# B&R Automation Studio project DuctLines (part 15)

### Program Logical/Uncoiler_2 (IEC)

#### Cyclic.ld - Cyclic code
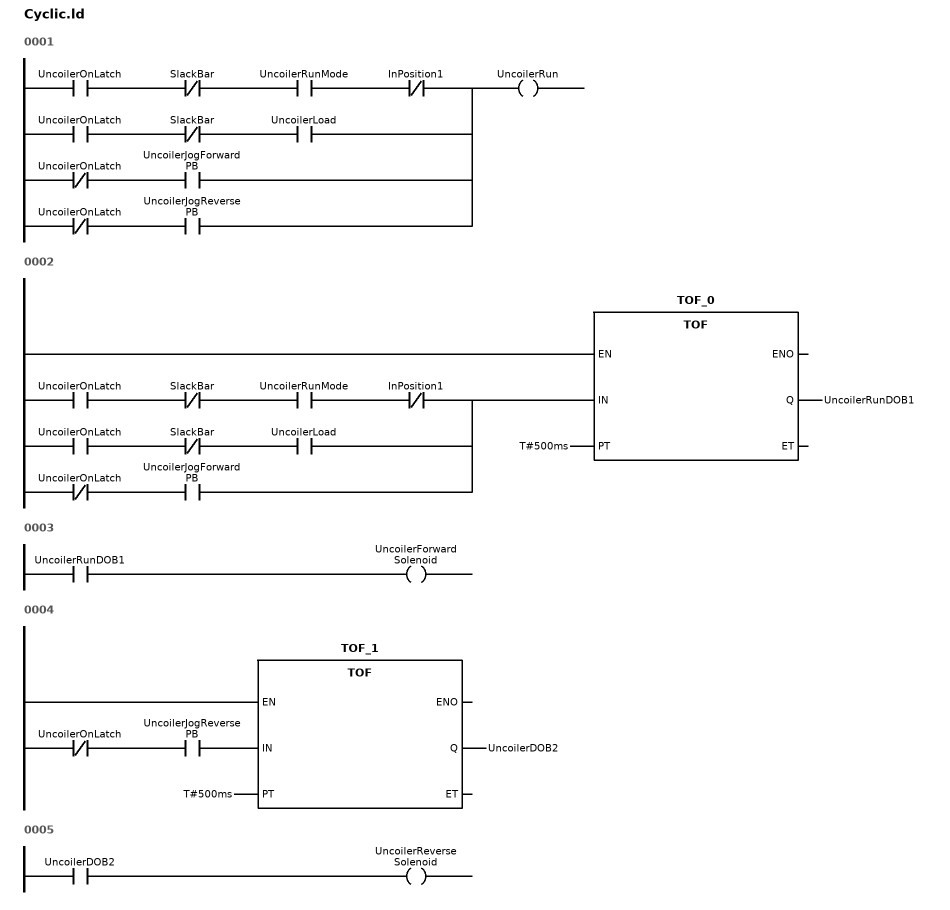
Ladder, written as Structured Text:
```iecst
PROGRAM _CYCLIC
(* Network 1 *)
UncoilerRun := (UncoilerOnLatch AND NOT SlackBar AND ((UncoilerRunMode AND NOT InPosition1) OR UncoilerLoad)) OR (NOT UncoilerOnLatch AND (UncoilerJogForwardPB OR UncoilerJogReversePB));

(* Network 2 *)
TOF_0(IN := (UncoilerOnLatch AND NOT SlackBar AND ((UncoilerRunMode AND NOT InPosition1) OR UncoilerLoad)) OR (NOT UncoilerOnLatch AND UncoilerJogForwardPB), PT := T#500ms);
UncoilerRunDOB1 := TOF_0.Q;

(* Network 3 *)
UncoilerForwardSolenoid := UncoilerRunDOB1;

(* Network 4 *)
TOF_1(IN := NOT UncoilerOnLatch AND UncoilerJogReversePB, PT := T#500ms);
UncoilerDOB2 := TOF_1.Q;

(* Network 5 *)
UncoilerReverseSolenoid := UncoilerDOB2;
END_PROGRAM
```

#### Init.ld - Initialization code
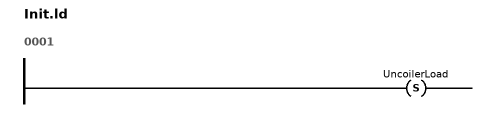
Ladder, written as Structured Text:
```iecst
PROGRAM _INIT
(* Network 1 *)
UncoilerLoad := TRUE;
END_PROGRAM
```

#### Variables.var - Local variables
```iecst
VAR
	TOF_0 : TOF;
	UncoilerRunDOB1 : BOOL;
	TOF_1 : TOF;
	UncoilerDOB2 : BOOL;
END_VAR
```

### Program Logical/IMotion1 (IEC) - Iowa Electric Servo Wrap Brake Routine 

#### Cyclic.st - Cyclic code
```iecst
PROGRAM _CYCLIC
	(*Iowa  Electric Servo Brake Motion Control*)
	IF ElectricWrapBrake THEN
		IF BrakeHydraulics AND BrakeDriveReady THEN
			IF NOT BrakeDriveEnable THEN
				BrakeDriveEnable := TRUE;
				MotionStatus2 := 0;
			END_IF;
		END_IF;
		IF NOT BrakeHydraulics THEN
			BrakeDriveEnable := FALSE;
		END_IF;
		IF NOT BrakeDriveReady THEN
			BrakeDriveEnable := FALSE;
		END_IF;
		IF NOT BrakeDriveEnable THEN
			MotionStatus2 := -1;
			ActualDAC2 := 0;
			StopFlag2 := 1;
			IMotion2Target := BrakeEncoder + IBrakeReference;
		END_IF;
		(*Brake Carriage Jogs*)
		IF BrakeDriveEnable AND NOT BrakeAuto THEN
			IF diBrakeCarriageJogIn THEN
				MotionStatus2 := 5;
			ELSE
				IF MotionStatus2 = 8 THEN
					StopFlag2 := 1;
				END_IF;
			END_IF; (*Jog In*)
			IF diBrakeCarriageJogOut THEN
				MotionStatus2 := 4;
			ELSE
				IF MotionStatus2 = 7 THEN
					StopFlag2 := 1;
				END_IF;
			END_IF; (*Jog Out*)
		END_IF; (*Jogs*)
	END_IF;	(*Electric Wrap Brake*)
	difference := IMotion2Target - (BrakeEncoder + IBrakeReference);
	AbsoluteDifference := ABS(difference);
	CASE MotionStatus2 OF
		(*Hold Position*)
		0:
			IF NOT InPosition2 THEN
				IF AbsoluteDifference <= BrakeTolerance THEN
					TargetCount2 := TargetCount2 + UpdateRate2;
					IF TargetCount2 >= SettleTime2 THEN
						InPosition2 := TRUE;
					END_IF;
				END_IF;
			END_IF;

			IF (difference * 6) < MaxDAC THEN
				Ratio2 := DINT_TO_INT(difference * 10); (*Was 15 *)
			ELSE
				Ratio2 := 15000;
		    END_IF;
			IF Counter2 > 0 THEN
				Counter2 := Counter2 - UpdateRate2;
			ELSE
				Counter2 := 500;
				IF Hold2 <> Ratio2 THEN
					Hold2 := Ratio2;
				ELSE
					DACBalance2 := ActualDAC2;
				END_IF;
			END_IF;

			TargetDAC2 := Ratio2 + DACBalance2;
			ActualDAC2 := TargetDAC2;

			IF ActualDAC2 > TopDAC2 THEN
				ActualDAC2 := TopDAC2;
			END_IF;
			IF ActualDAC2 < -TopDAC2 THEN
				ActualDAC2 := -TopDAC2;
			END_IF

		(*Initialize Move*)
		1:
			Axis2Scaler := (BrakeDesired / BrakeActual);
			IMotion2Target := REAL_TO_DINT(BrakeCarriageTarget * BrakeResolution * Axis2Scaler);
			IBrakeReference := REAL_TO_DINT(BrakeReference * BrakeResolution * Axis2Scaler);
			DACAdd2 := INT_TO_REAL(MaxDAC) / AccelRampReal2;
			ActualSpeed2 := (TopAxis2Speed * DINT_TO_REAL(BrakePercentSpeed)) / 100.0; (*Real Counts Per Second*)
			ActualRunPercent2 := DINT_TO_REAL(BrakePercentSpeed) / 100.0;
			TopDAC2 := REAL_TO_INT(INT_TO_REAL(MaxDAC) * ActualRunPercent2);
			IF ActualRunPercent2 = 1.0 THEN
				TopDAC2 := TopDAC2 - REAL_TO_INT(INT_TO_REAL(UpdateRate2) * DACAdd2);
			END_IF;
			AverageSpeed2 := ActualSpeed2 / 2.0;
			DecelTime2 := (DecelRampReal2 / 1000.0) * ActualRunPercent2;
			DecelDistance2 := REAL_TO_DINT((AverageSpeed2 * DecelTime2 ) * Axis2Scaler);
			SRM2 := MaxDACSquared / ((TopAxis2Speed * (AccelRampReal2 / 1000.0)) / 2.0);
			MoveLength2 := IMotion2Target - (BrakeEncoder + IBrakeReference);
			AMoveLength2 := ABS(MoveLength2);
			IF DecelDistance2 > (AMoveLength2 / 2) THEN
				DecelDistance2 := AMoveLength2 / 2;
				TopDAC2 := REAL_TO_INT(SQRT((DINT_TO_REAL(DecelDistance2) / Axis2Scaler) * SRM2));
				IF TopDAC2 < 3276 THEN
					TopDAC2 := 3276;
				END_IF;
			END_IF;
			InPosition2 := FALSE;
			FirstTarget2 := FALSE;
			StopWatch2 := 0.0;
			IF AMoveLength2 > REAL_TO_DINT(BrakeResolution / 16.0) THEN
				IF MoveLength2 >= 0 THEN
				  MotionStatus2 := 2;
			    ELSE
				  MotionStatus2 := 10;
				END_IF;
			ELSE
				MotionStatus2 := 12;
		    END_IF;
		(*Ramp Up To Speed*)
		2:
			IF DecelDistance2 < difference THEN
				ActualDAC2 := ActualDAC2 + REAL_TO_INT(INT_TO_REAL(UpdateRate2) * DACAdd2);
				IF ActualDAC2 > TopDAC2 THEN
					ActualDAC2 := TopDAC2;
				END_IF;
			ELSE (*Switch To Decel MotionState*)
				DecelCounter2 := 200;
				LastPosition2 := BrakeEncoder;
				TargetCount2 := 0;
				FirstTarget2 := FALSE;
				MotionStatus2 := 3;
			END_IF;
		3: (*Decel To Target*)
			(*Stall Detection*)
			DecelCounter2 := DecelCounter2 - UpdateRate2;
			IF DecelCounter2 <= 0 THEN
				DecelCounter2 := 200;
				IF LastPosition2 = BrakeEncoder THEN
					DACBalance2 := ActualDAC2;
					Counter2 := 500;
					TopDAC2 := MaxDAC / 4;
					MotionStatus2 := 0;
				ELSE
					LastPosition2 := BrakeEncoder;
				END_IF;
			END_IF;

			RealDAC2 := REAL_TO_INT(SQRT(DINT_TO_REAL(AbsoluteDifference) * SRM2));
			IF RealDAC2 > INT_TO_REAL(MaxDAC) THEN
				RealDAC2 := INT_TO_REAL(MaxDAC);
			END_IF;
			ActualDAC2 := REAL_TO_INT(RealDAC2);

			IF FirstTarget2 THEN
				(*ActualDAC2 := ActualDAC2 / 8;*)
			END_IF;

			IF difference < 0 THEN
				ActualDAC2 := -ActualDAC2;
			END_IF;

			IF AbsoluteDifference <= BrakeTolerance THEN
				FirstTarget2 := TRUE;
				TargetCount2 := TargetCount2 + UpdateRate2;
				IF TargetCount2 >= SettleTime2 THEN
					Counter2 := 500;
					InPosition2 := TRUE;
					MotionStatus2 := 0;
					TopDAC2 := MaxDAC / 4;
				END_IF;
			ELSE
				TargetCount2 := 0;
			END_IF;
		4: (*Setup Forward Jog*)
			DACAdd2 := INT_TO_REAL(MaxDAC) / AccelRampReal2;
			TopDAC2 := DINT_TO_INT((INT_TO_DINT(MaxDAC) * BackGaugeJogPercent) / 100);
			TopDAC2 := TopDAC2 - REAL_TO_INT(DACAdd2);
			IBrakeReference := REAL_TO_DINT(BrakeReference * BrakeResolution * Axis2Scaler);
			StopFlag2 := FALSE;
			MotionStatus2 := 7;
		5: (*Setup Reverse Jog*)
			DACAdd2 := INT_TO_REAL(MaxDAC) / AccelRampReal2;
			TopDAC2 := DINT_TO_INT((INT_TO_DINT(MaxDAC) * BackGaugeJogPercent) / 100);
			TopDAC2 := TopDAC2 - REAL_TO_INT(DACAdd2);
			IBrakeReference := REAL_TO_DINT(BrakeReference * BrakeResolution * Axis2Scaler);
			StopFlag2 := FALSE;
			InPosition1 := FALSE;
			MotionStatus2 := 8;
		7: (*Forward Jog*)
			IF CarriageReference THEN
				StopFlag2 := 1;
			END_IF;
			IF StopFlag2 THEN
				IF ActualDAC2 > REAL_TO_INT(DACAdd2) THEN (*Decelerate*)
					ActualDAC2 := ActualDAC2 - REAL_TO_INT(DACAdd2);
				ELSE (*Hold Position*)
					ActualDAC2 := 0;
					IMotion2Target := BrakeEncoder + IBrakeReference;
					InPosition2 := TRUE;
					MotionStatus2 := 0;
				END_IF;
			ELSE
				InPosition2 := FALSE;
				IF ActualDAC2 < TopDAC2 THEN (*Accelerate*)
					ActualDAC2 := ActualDAC2 + REAL_TO_INT(DACAdd2);
				ELSE
					ActualDAC2 := TopDAC2; (*Maintain Constant Speed*)
				END_IF;
			END_IF;
		8: (*Reverse Jog*)
			IF EjectComplete THEN
				StopFlag2 := TRUE;
			END_IF;
			IF StopFlag2 THEN
				IF ActualDAC2 < REAL_TO_INT(-DACAdd2) THEN (*Decelerate*)
					ActualDAC2 := ActualDAC2 + REAL_TO_INT(DACAdd2);
				ELSE (*Hold Position*)
					ActualDAC2 := 0;
					IMotion2Target := BrakeEncoder + IBrakeReference;
					InPosition2 := TRUE;
					MotionStatus2 := 0;
				END_IF;
			ELSE
				IF ActualDAC2 > -TopDAC2 THEN (*Accelerate*)
					ActualDAC2 := ActualDAC2 - REAL_TO_INT(DACAdd2);
				ELSE
					ActualDAC2 := -TopDAC2; (*Maintain Constant Speed*)
				END_IF;
			END_IF;
		9:
			IF ActualDAC2 > REAL_TO_INT(DACAdd1) THEN (*Decelerate*)
				ActualDAC2 := ActualDAC2 - REAL_TO_INT(DACAdd2);
			ELSE (* Hold Position *)
				MetalTarget := ActlMetalEncoder;
				IncrementalRealTarget := DINT_TO_REAL(difference) / UnitsPerInch1 / MetalScaler;
				MotionStatus1 := 0;
			END_IF;
		10:
			IF DecelDistance2 < AbsoluteDifference THEN
				ActualDAC2 := ActualDAC2 - REAL_TO_INT(INT_TO_REAL(UpdateRate2) * DACAdd2);
				IF ActualDAC2 < -TopDAC2 THEN
					ActualDAC2 := -TopDAC2;
				END_IF;
			ELSE (*Switch To Decel MotionState*)
				DecelCounter2 := 200;
				LastPosition2 := BrakeEncoder;
				TargetCount2 := 0;
				FirstTarget2 := FALSE;
				MotionStatus2 := 3;
			END_IF;
		12:
			StopWatch2 := StopWatch2 + INT_TO_REAL(UpdateRate2);
			IF StopWatch2 > 100 THEN
				InPosition2 := TRUE;
				MotionStatus2 := 0;
			END_IF;
		ELSE (*Not Moving Or Holding*)
			ActualDAC2 := 0;
			IMotion2Target := BrakeEncoder + IBrakeReference;
			InPosition2 := TRUE;
	END_CASE;

	IF ActualDAC2 > MaxDAC THEN
		ActualDAC2 := MaxDAC;
	END_IF;
	IF ActualDAC2 < -MaxDAC THEN
		ActualDAC2 := -MaxDAC;
	END_IF;

END_PROGRAM
```

#### Variables.var - Local variables
```iecst
VAR
	AbsoluteDifference : DINT;
	ActualRunPercent2 : REAL;
	ActualSpeed2 : REAL;
	AMoveLength2 : DINT;
	AverageSpeed2 : REAL;
	Axis2Scaler : REAL;
	Counter2 : INT;
	DACAdd2 : REAL;
	DACBalance2 : INT;
	DecelCounter2 : INT;
	DecelDistance2 : DINT;
	DecelTime2 : REAL;
	difference : DINT;
	FirstTarget2 : BOOL;
	Hold2 : INT;
	LastPosition2 : DINT;
	MoveLength2 : DINT;
	Ratio2 : INT;
	RealDAC2 : REAL;
	SRM2 : REAL;
	StopWatch2 : REAL;
	TargetCount2 : INT;
	TargetDAC2 : INT;
	TopAxis2Speed : REAL := 204800;
	TopDAC2 : INT;
END_VAR
```

### Program Logical/MarkHead (IEC)

#### Variables.var
```iecst
VAR
	Dn1Delay : BOOL;
	Dn1Done : BOOL;
	Dn1Latch : BOOL;
	Dn2Latch : BOOL;
	PassUpPulse : BOOL;
	TON_0 : TON;
	TON_10ms_0 : TON_10ms;
	TON_10ms_1 : TON_10ms;
	TPulseLength : TIME := T#10s;
	TP_0 : TP;
	TP_1 : TP;
	TP_2 : TP;
	TP_10ms_0 : TP_10ms;
	Up1Latch : BOOL;
	Up2Done : BOOL;
	Up2Latch : BOOL;
	Up2PassLatch1 : BOOL;
END_VAR
```

#### Cyclic.ld
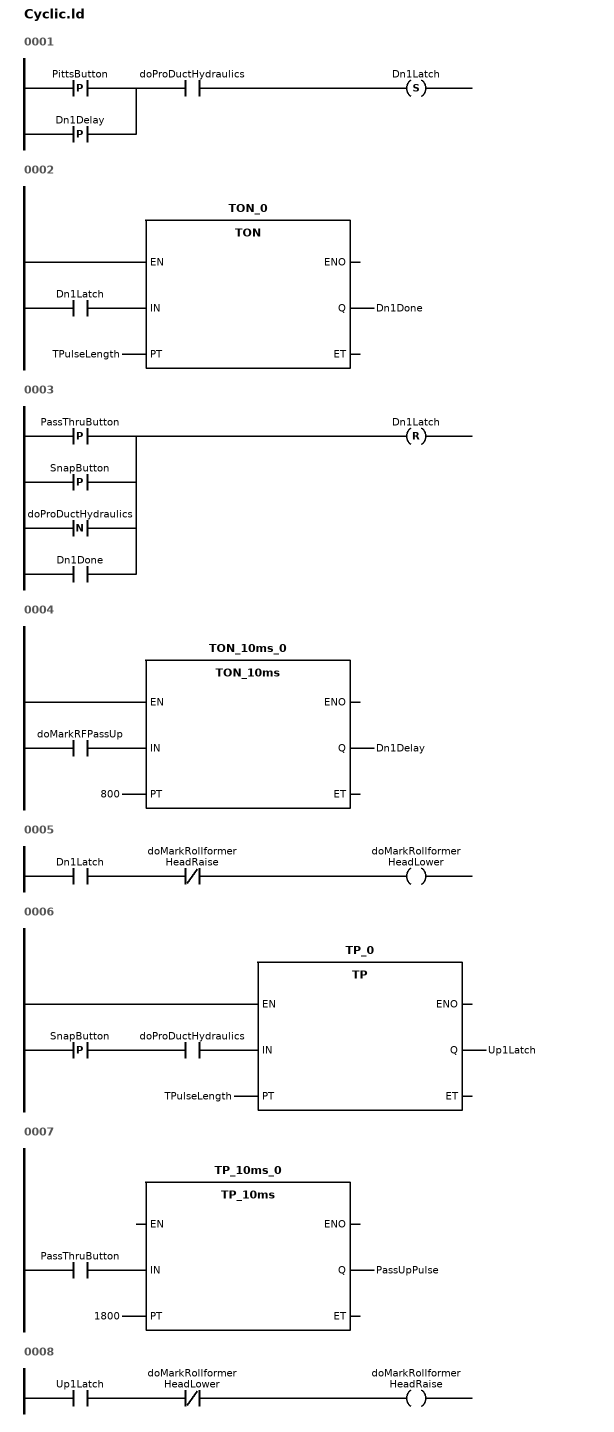
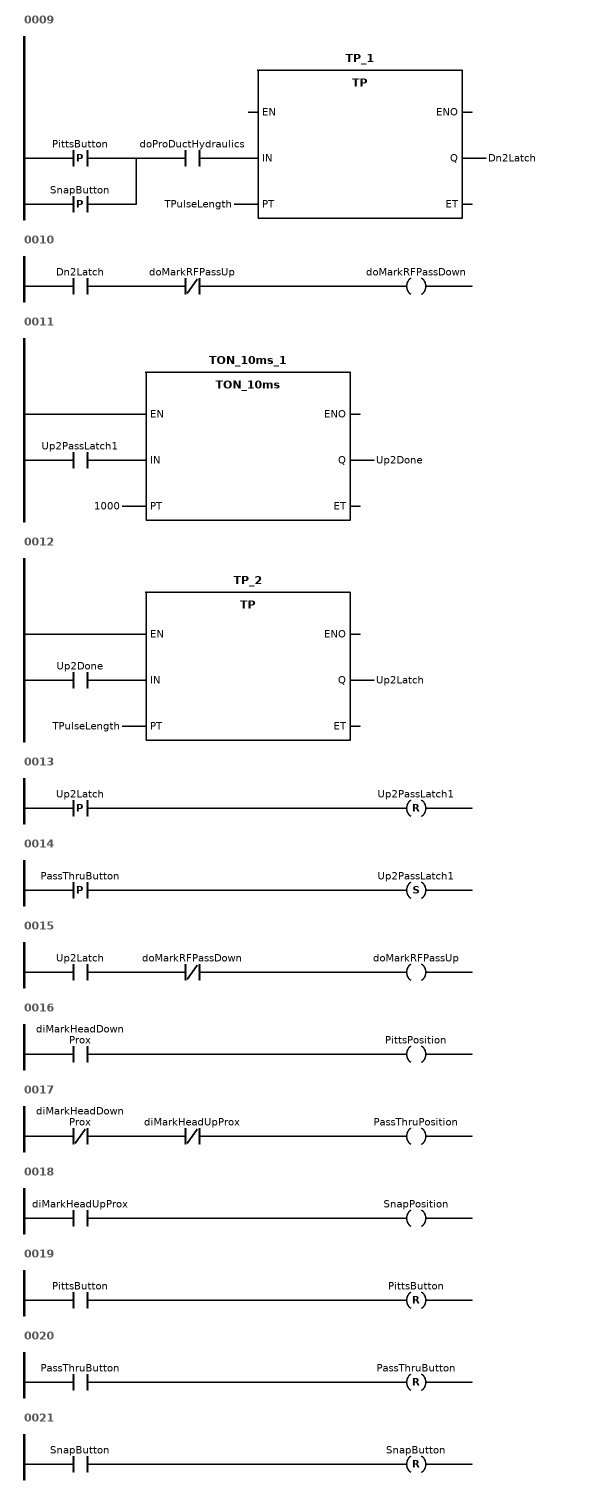
Ladder, written as Structured Text:
```iecst
PROGRAM _CYCLIC
VAR
    _e1 : R_TRIG;
    _e2 : R_TRIG;
    _e3 : R_TRIG;
    _e4 : R_TRIG;
    _e5 : F_TRIG;
    _e6 : R_TRIG;
    _e7 : R_TRIG;
    _e8 : R_TRIG;
    _e9 : R_TRIG;
    _e10 : R_TRIG;
END_VAR
(* Network 1 *)
_e1(CLK := PittsButton);
_e2(CLK := Dn1Delay);
IF (_e1.Q OR _e2.Q) AND doProDuctHydraulics THEN Dn1Latch := TRUE; END_IF;

(* Network 2 *)
TON_0(IN := Dn1Latch, PT := TPulseLength);
Dn1Done := TON_0.Q;

(* Network 3 *)
_e3(CLK := PassThruButton);
_e4(CLK := SnapButton);
_e5(CLK := doProDuctHydraulics);
IF _e3.Q OR _e4.Q OR _e5.Q OR Dn1Done THEN Dn1Latch := FALSE; END_IF;

(* Network 4 *)
TON_10ms_0(IN := doMarkRFPassUp, PT := 800);
Dn1Delay := TON_10ms_0.Q;

(* Network 5 *)
doMarkRollformerHeadLower := Dn1Latch AND NOT doMarkRollformerHeadRaise;

(* Network 6 *)
_e6(CLK := SnapButton);
TP_0(IN := _e6.Q AND doProDuctHydraulics, PT := TPulseLength);
Up1Latch := TP_0.Q;

(* Network 7 *)
TP_10ms_0(IN := PassThruButton, PT := 1800);
PassUpPulse := TP_10ms_0.Q;

(* Network 8 *)
doMarkRollformerHeadRaise := Up1Latch AND NOT doMarkRollformerHeadLower;

(* Network 9 *)
_e7(CLK := PittsButton);
_e8(CLK := SnapButton);
TP_1(IN := (_e7.Q OR _e8.Q) AND doProDuctHydraulics, PT := TPulseLength);
Dn2Latch := TP_1.Q;

(* Network 10 *)
doMarkRFPassDown := Dn2Latch AND NOT doMarkRFPassUp;

(* Network 11 *)
TON_10ms_1(IN := Up2PassLatch1, PT := 1000);
Up2Done := TON_10ms_1.Q;

(* Network 12 *)
TP_2(IN := Up2Done, PT := TPulseLength);
Up2Latch := TP_2.Q;

(* Network 13 *)
_e9(CLK := Up2Latch);
IF _e9.Q THEN Up2PassLatch1 := FALSE; END_IF;

(* Network 14 *)
_e10(CLK := PassThruButton);
IF _e10.Q THEN Up2PassLatch1 := TRUE; END_IF;

(* Network 15 *)
doMarkRFPassUp := Up2Latch AND NOT doMarkRFPassDown;

(* Network 16 *)
PittsPosition := diMarkHeadDownProx;

(* Network 17 *)
PassThruPosition := NOT diMarkHeadDownProx AND NOT diMarkHeadUpProx;

(* Network 18 *)
SnapPosition := diMarkHeadUpProx;

(* Network 19 *)
IF PittsButton THEN PittsButton := FALSE; END_IF;

(* Network 20 *)
IF PassThruButton THEN PassThruButton := FALSE; END_IF;

(* Network 21 *)
IF SnapButton THEN SnapButton := FALSE; END_IF;
END_PROGRAM
```

### Program Logical/EFeeder_Junk

#### Variables.var
```iecst
VAR
	AnalogForward : BOOL;
	AnalogReverse : BOOL;
	AutoSignal : BOOL;
	BatchCancelUnlatch : BOOL;
	BeadRollFires : BOOL;
	BeadRollUsedUp : BOOL;
	Block_1 : BOOL;
	ButtonBack7 : BOOL;
	ButtonFires : BOOL;
	ButtonUsedUp : BOOL;
	CenterHoleFires : BOOL;
	CenterHoleTime : TIME;
	CenterHoleUsedUp : BOOL;
	CenterPosA : BOOL;
	CenterShuttleIndex : INT;
	ChangeCShuttle : BOOL;
	ChangeJob1 : BOOL;
	ChangeLShuttle : BOOL;
	ChangeRShuttle : BOOL;
	ClearEncoderSignal : BOOL;
	CleatFires : BOOL;
	CleatUsedUp : BOOL;
	CLPUnlatch : BOOL;
	CShuttleUnlatch : BOOL;
	CustomLTFires : BOOL;
	CustomLTTime : TIME;
	CustomLTUsedUp : BOOL;
	CustomLTValve : BOOL;
	CustomVFires : BOOL;
	CustomVTime : TIME;
	CustomVUsedUp : BOOL;
	DamperLatch : BOOL;
	DamperResult : DINT;
	DataUpdated : BOOL;
	DDDoneTimer : TON;
	DieDelayDone : BOOL;
	DieUpTime : TIME;
	DirectionDelayDone : BOOL;
	DuctoAutoUnlatch : BOOL;
	FFCLatch : BOOL;
	FiveFootCoil : BOOL;
	FourFootCoil : BOOL;
	FourResult : DINT;
	GapPulse : BOOL;
	GapTP : BOOL;
	GTime : TIME;
	HalfUpdated1 : BOOL;
	HalfUpdated2 : BOOL;
	HolePunchSelecedtSolenoid : BOOL;
	IncPartsMade : BOOL;
	InitMoveSignal : BOOL;
	InPositionBand : REAL := 0.01;
	JobChanging : BOOL;
	LeftHoleFires : BOOL;
	LeftHoleTime : TIME;
	LeftHoleUsedUp : BOOL;
	LeftPosA : BOOL;
	LShuttleUnlatch : BOOL;
	LTFires : BOOL;
	LTTime : TIME;
	LTUsedUp : BOOL;
	ManualSignal : BOOL;
	MarkAccumulator : REAL;
	MetalEncoderLatch : DINT;
	NewRunJobOk : BOOL;
	NextMoveComplete : BOOL;
	NextMoveLookAgain : BOOL;
	NoShearHits : BOOL;
	OGLatch : BOOL;
	OGResult : DINT;
	OneResult : DINT;
	OutsideLatch : BOOL;
	PartCutOff : BOOL;
	PartRefOK : BOOL;
	PunchCurrentSelect : DINT;
	RightHoleFires : BOOL;
	RightHoleTime : TIME;
	RightHoleUsedUp : BOOL;
	RightPosA : BOOL;
	RollEnableUnlatch : BOOL;
	RShuttleUnlatch : BOOL;
	RTotalInches : REAL;
	RunSpeedCalculated : BOOL;
	SetConnectorChange : BOOL;
	ShearBrakeFires : BOOL;
	ShearBrakeUsedUp : BOOL;
	ShearFires : BOOL;
	ShearHitsLTZero : BOOL;
	shearTime : TIME;
	ShearUsedUp : BOOL;
	SixFootCoil : BOOL;
	SmallResult : REAL;
	Step04A : BOOL;
	Step05A : BOOL;
	Step05B : BOOL;
	Step06 : BOOL;
	Step07 : BOOL;
	Step08 : BOOL;
	Step09 : BOOL;
	Step10 : BOOL;
	Step15 : BOOL;
	Step16 : BOOL;
	Step17 : BOOL;
	Step18 : BOOL;
	Step18A : BOOL;
	Step18B : BOOL;
	Step19 : BOOL;
	ThirdOff1 : BOOL;
	ThirdOff2 : BOOL;
	ThirdOff3 : BOOL;
	TON_0 : TON;
	TON_1 : TON;
	TON_10 : TON;
	TON_Warning : TON;
	TP_0 : TP;
	TP_1 : TP;
	TP_2 : TP;
	TP_3 : TP;
	TP_4 : TP;
	TP_5 : TP;
	TP_6 : TP;
	TP_7 : TP;
	TP_8 : TP;
	TP_9 : TP;
	UnlatchBender : BOOL;
	UnlatchButtons : BOOL;
	VFires : BOOL;
	VTime : TIME;
	VUsedUp : BOOL;
	Wait1Ready : BOOL;
	Wait2Ready : BOOL;
	Wait3Ready : BOOL;
	WaitCon1 : BOOL;
	WaitCon2 : BOOL;
	ZCOLT0 : BOOL;
	ZCReverseComplete : BOOL;
	ZCSCTimer : TON;
	ZCSettleComplete : BOOL;
	ZeroCropDifference : DINT;
	ZRCTon : TON;
	FinalScan : BOOL;
	Step12 : BOOL;
	SHLT0 : BOOL;
	Step20 : BOOL;
	ReturnTarget : DINT;
	ReturnComplete : BOOL;
	Step21 : BOOL;
	ReturnCalculated : BOOL;
	Step22 : BOOL;
	JobsDifferent : BOOL;
END_VAR
```

#### Cyclic.ld
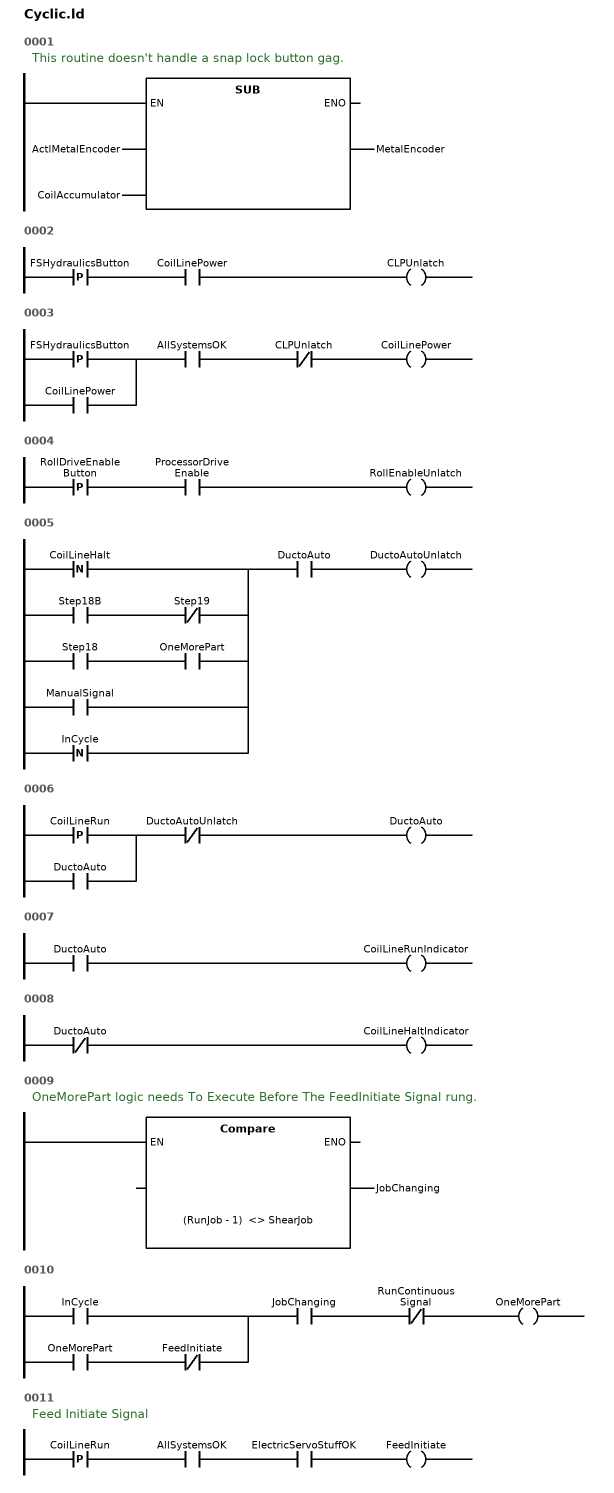
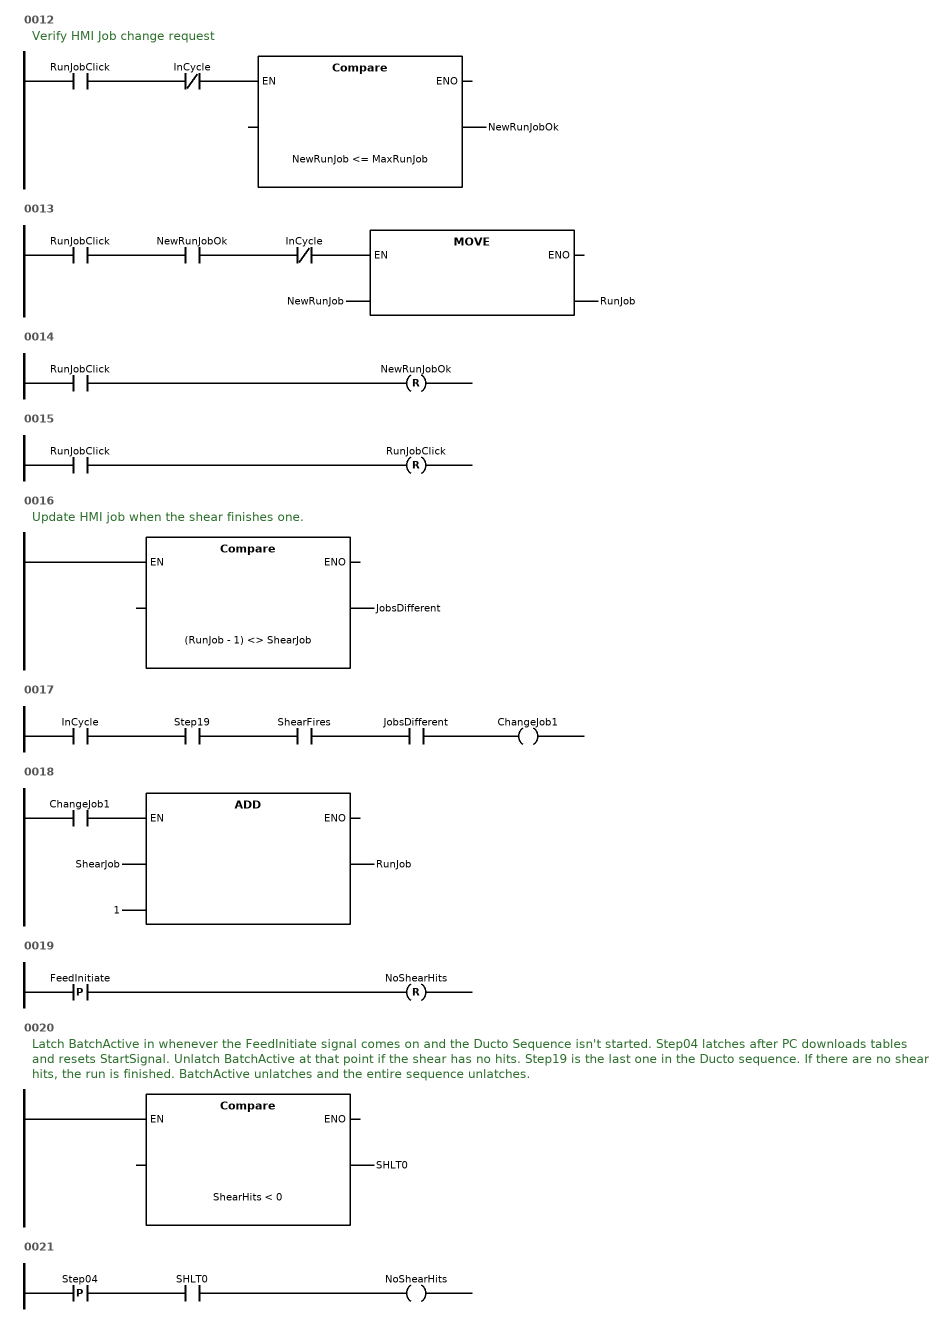
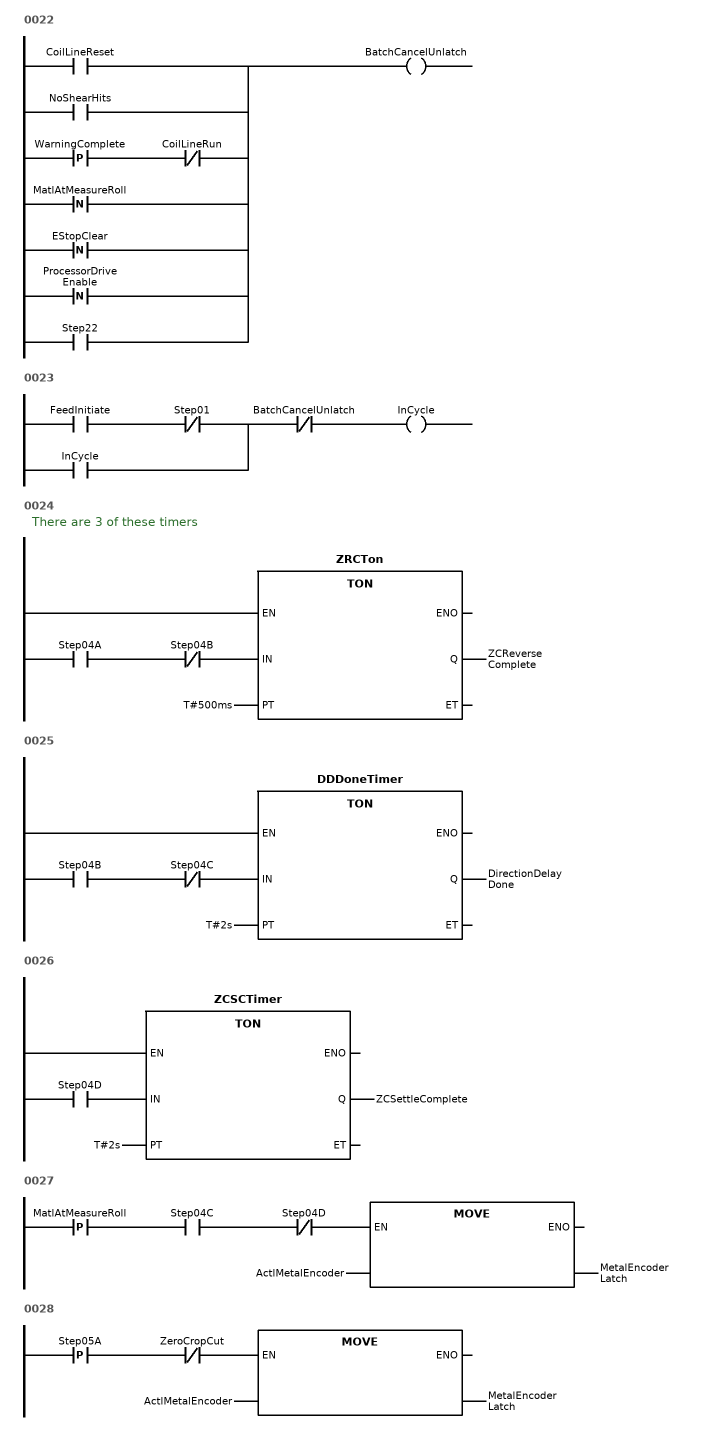
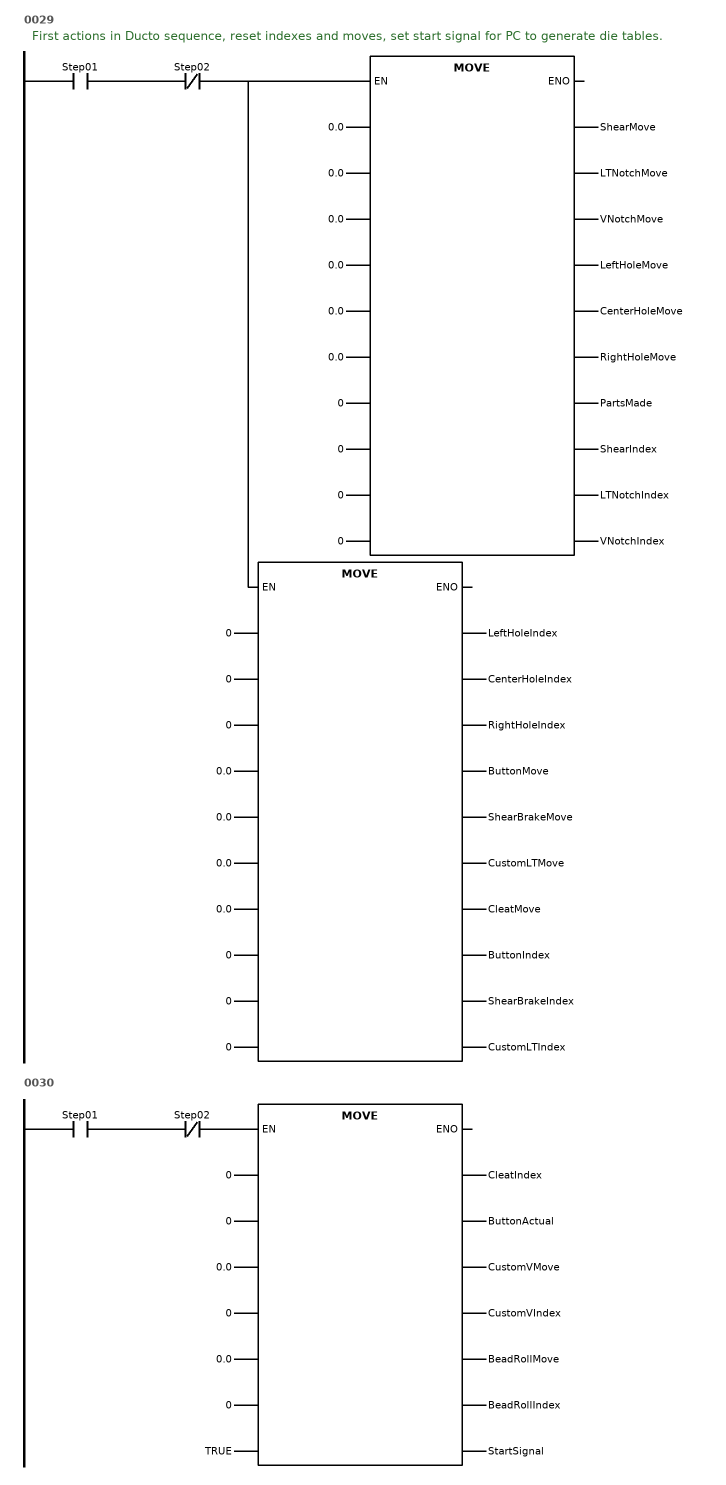
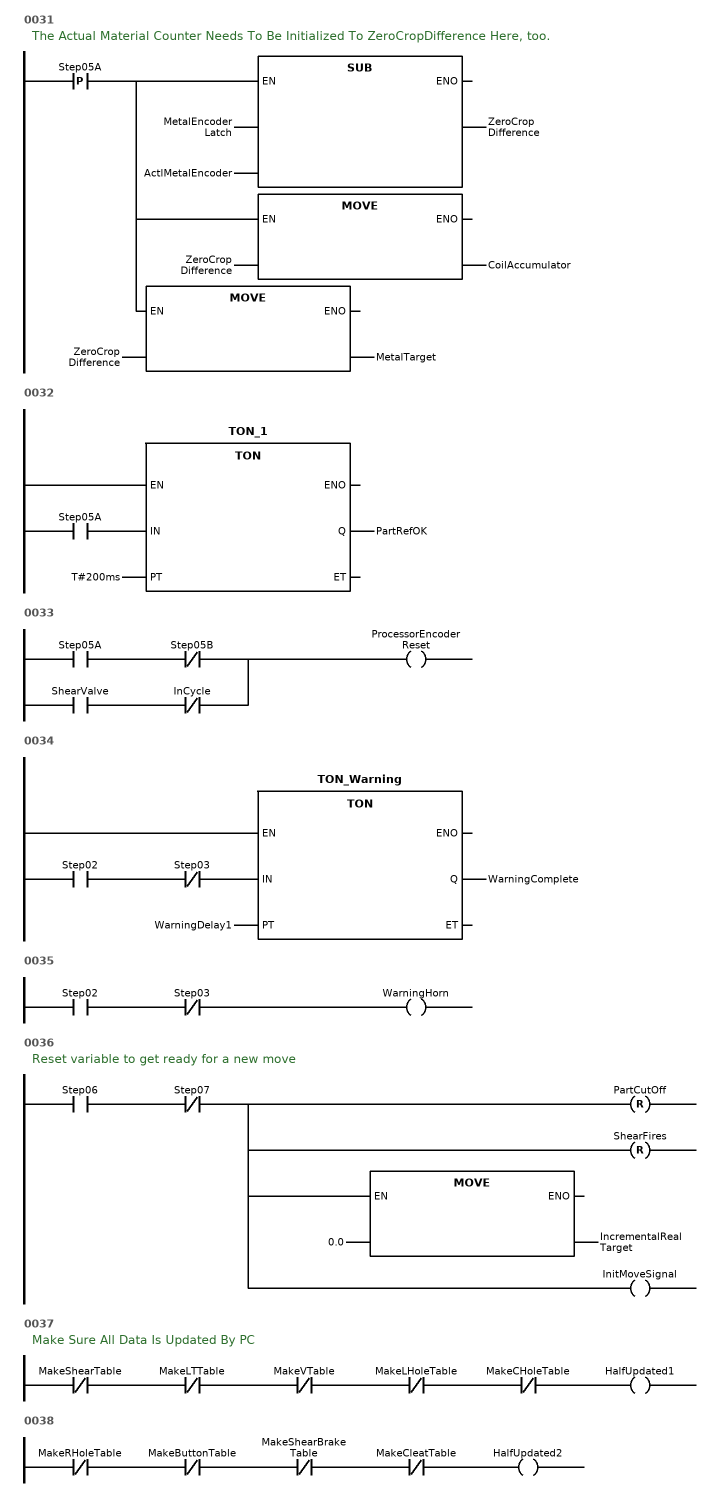
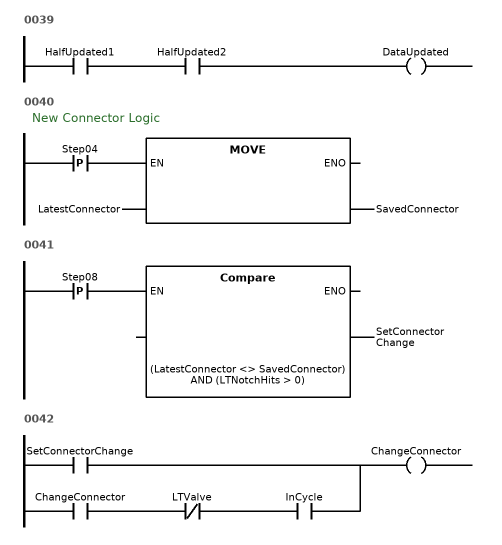
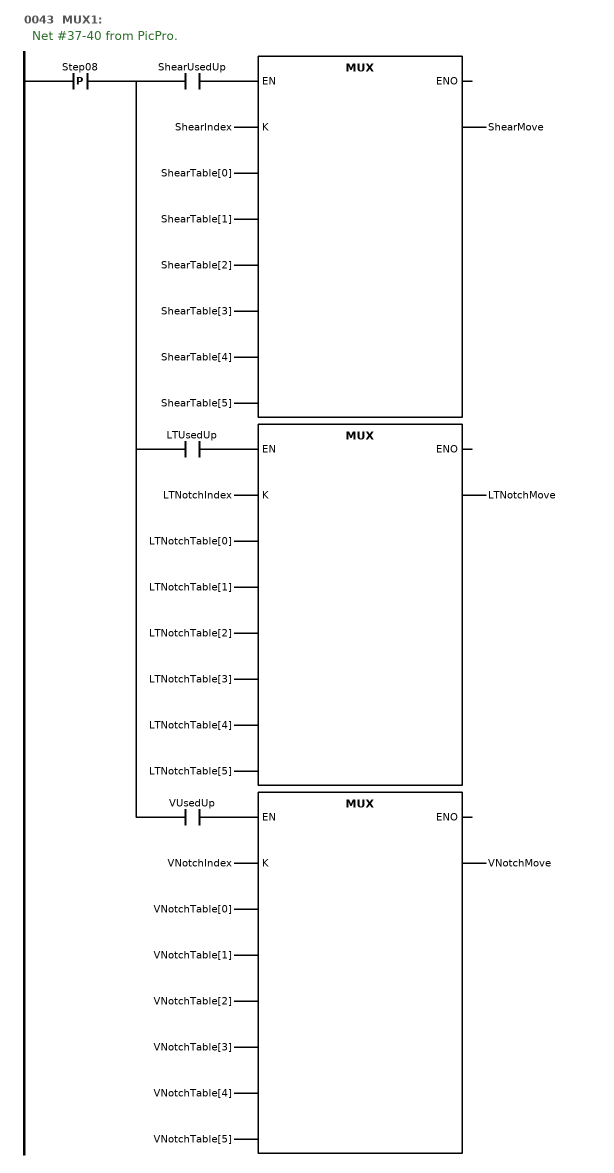
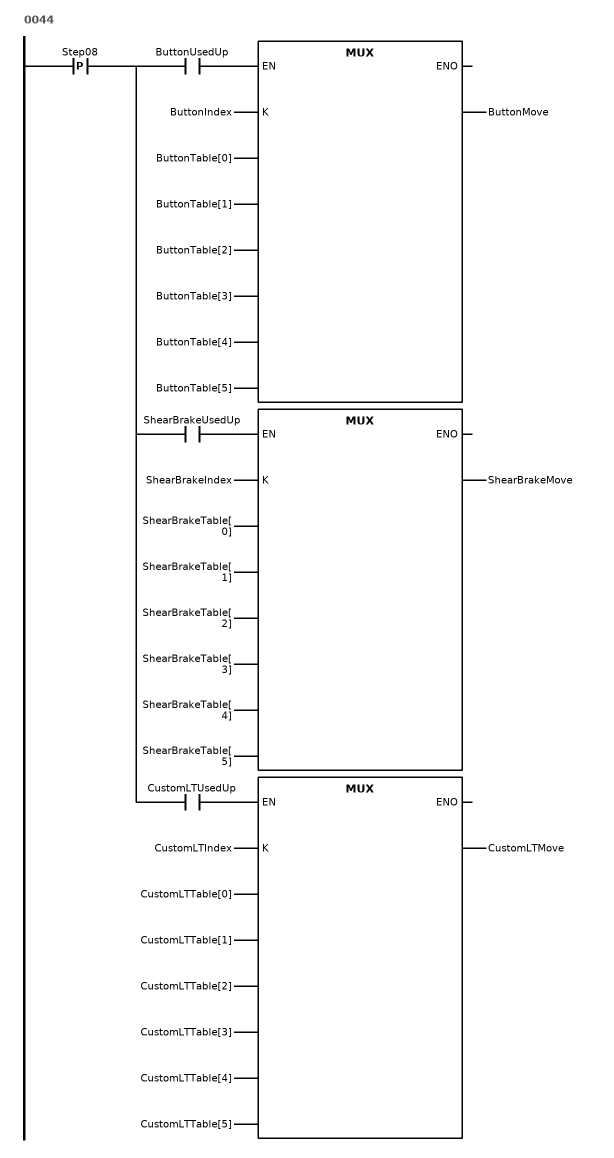
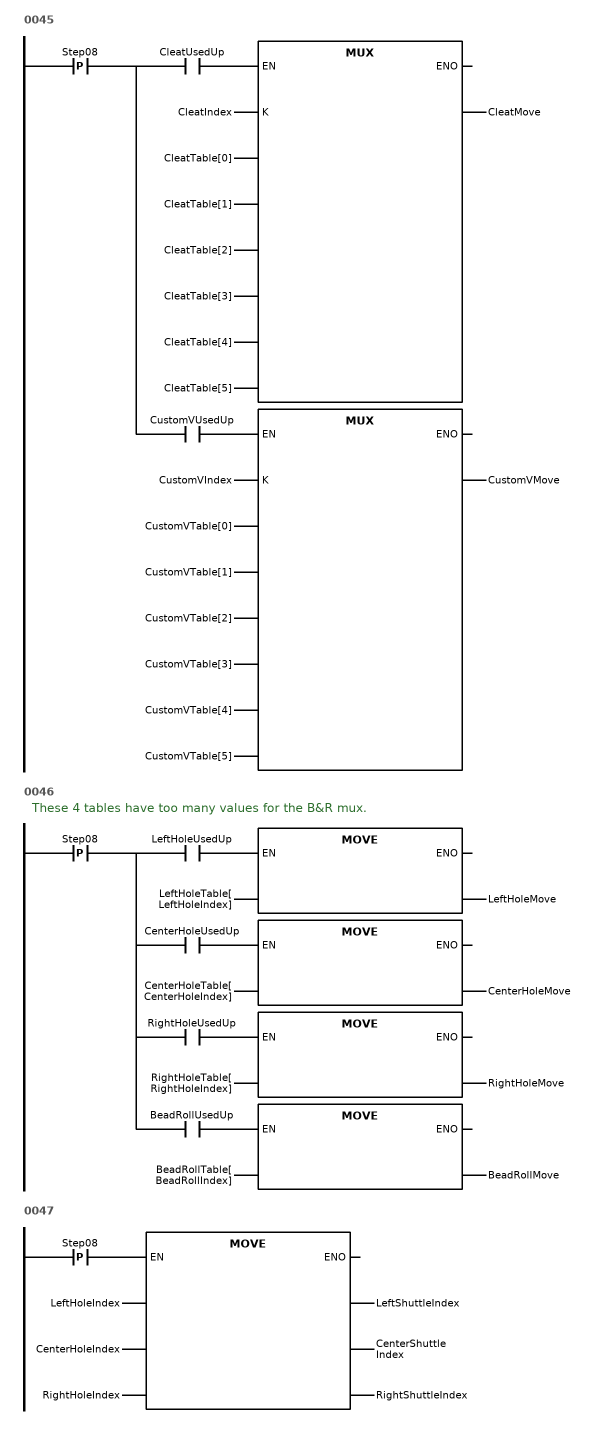
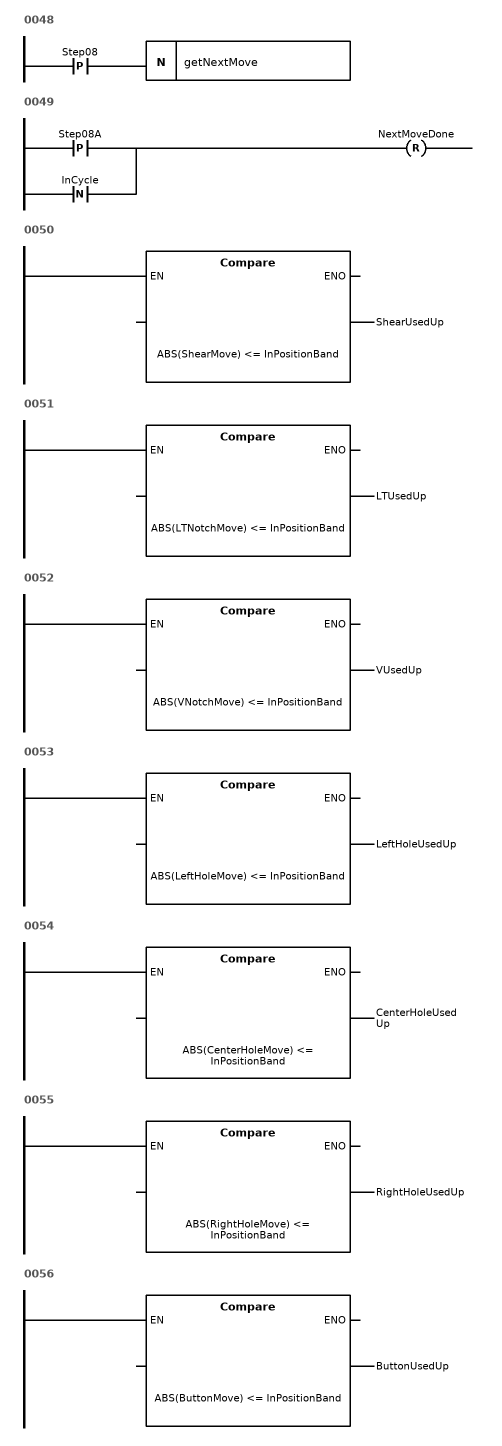
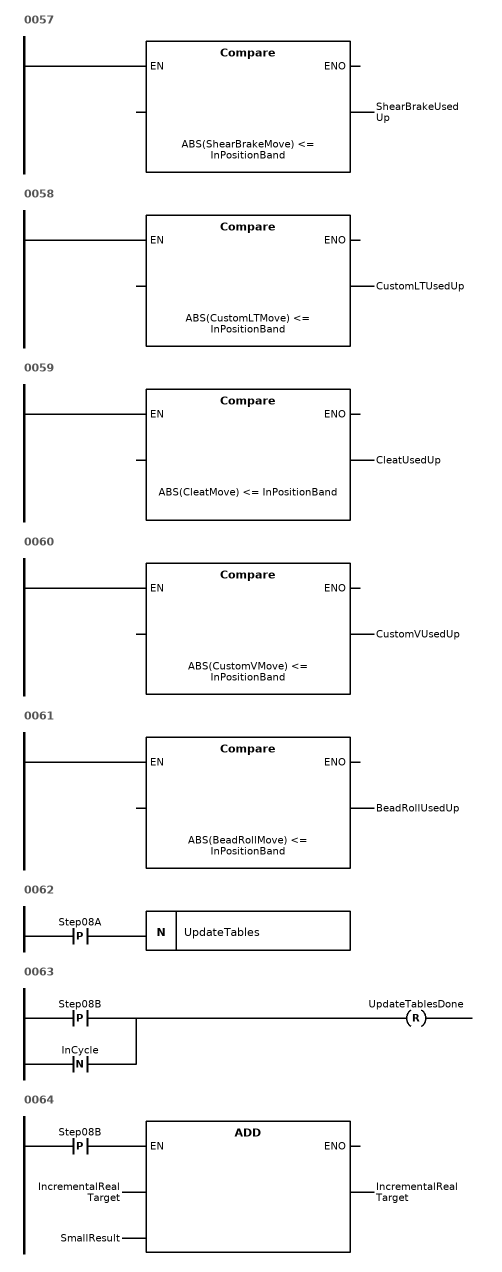
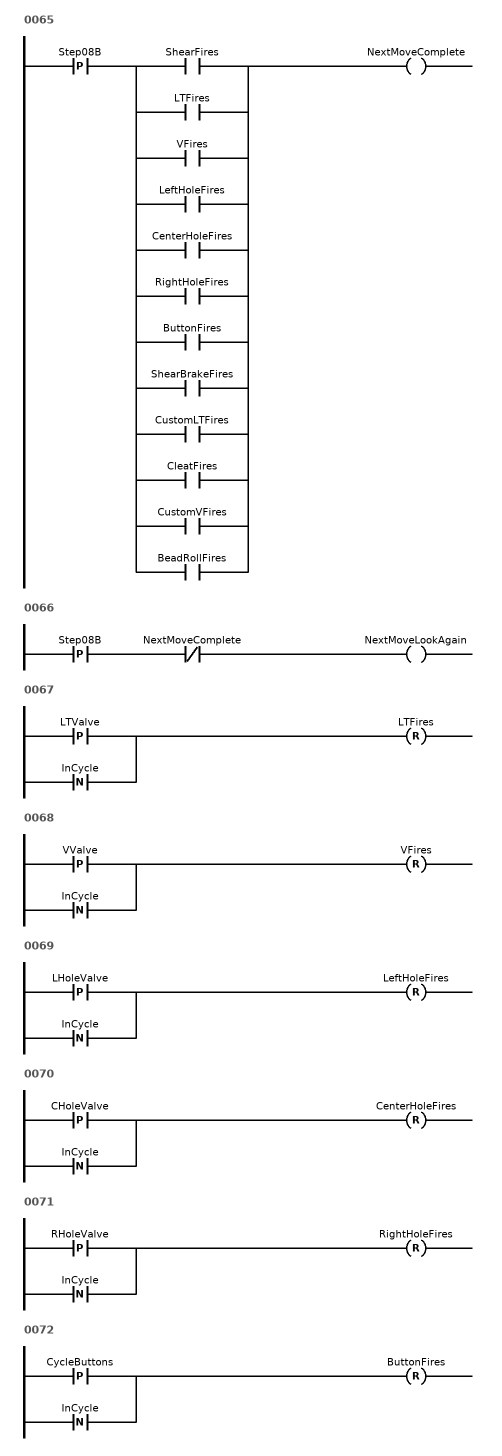
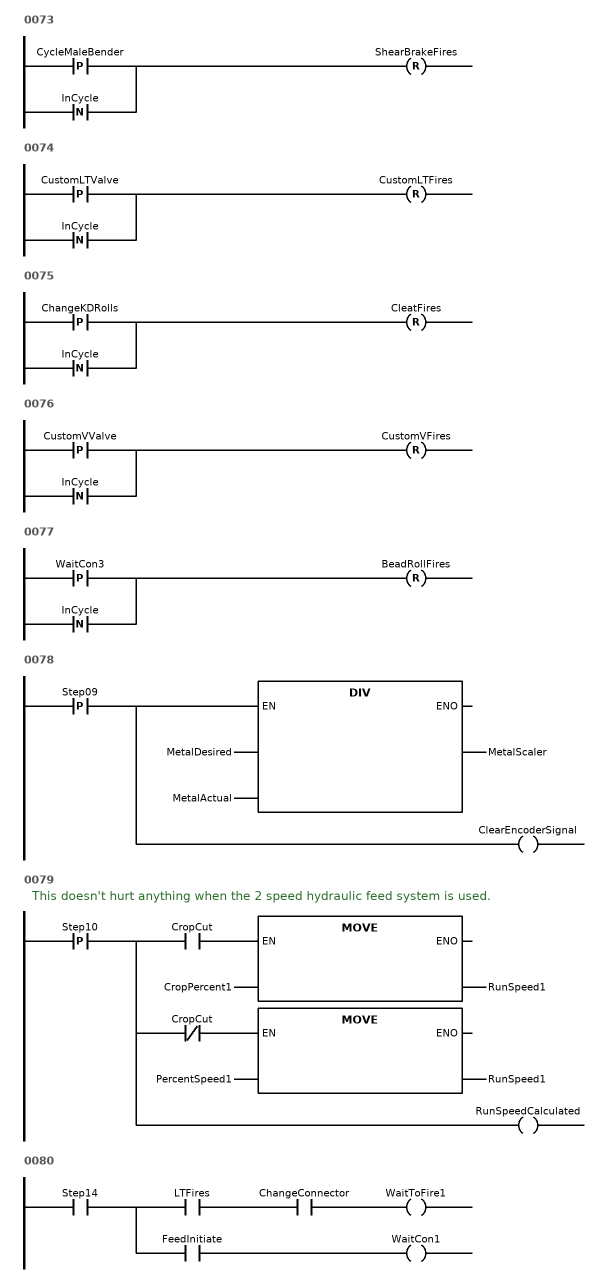
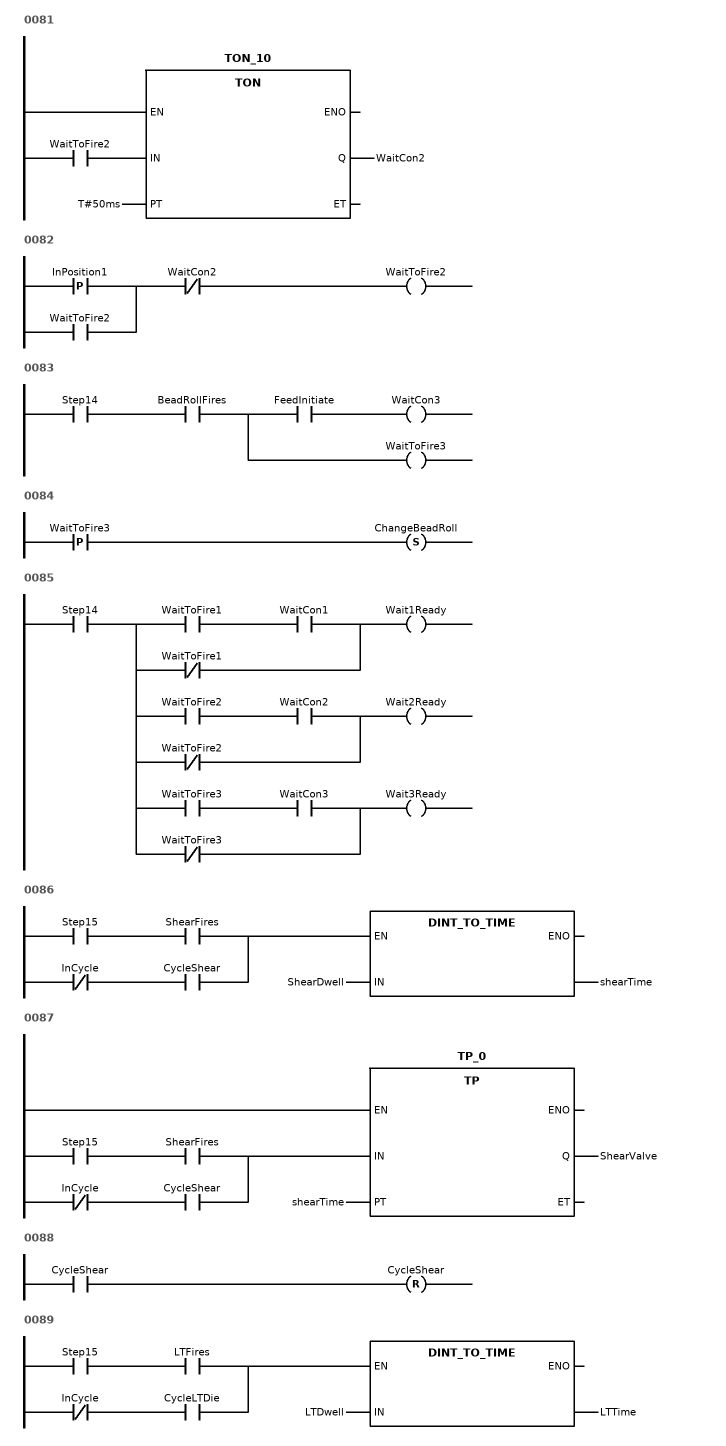
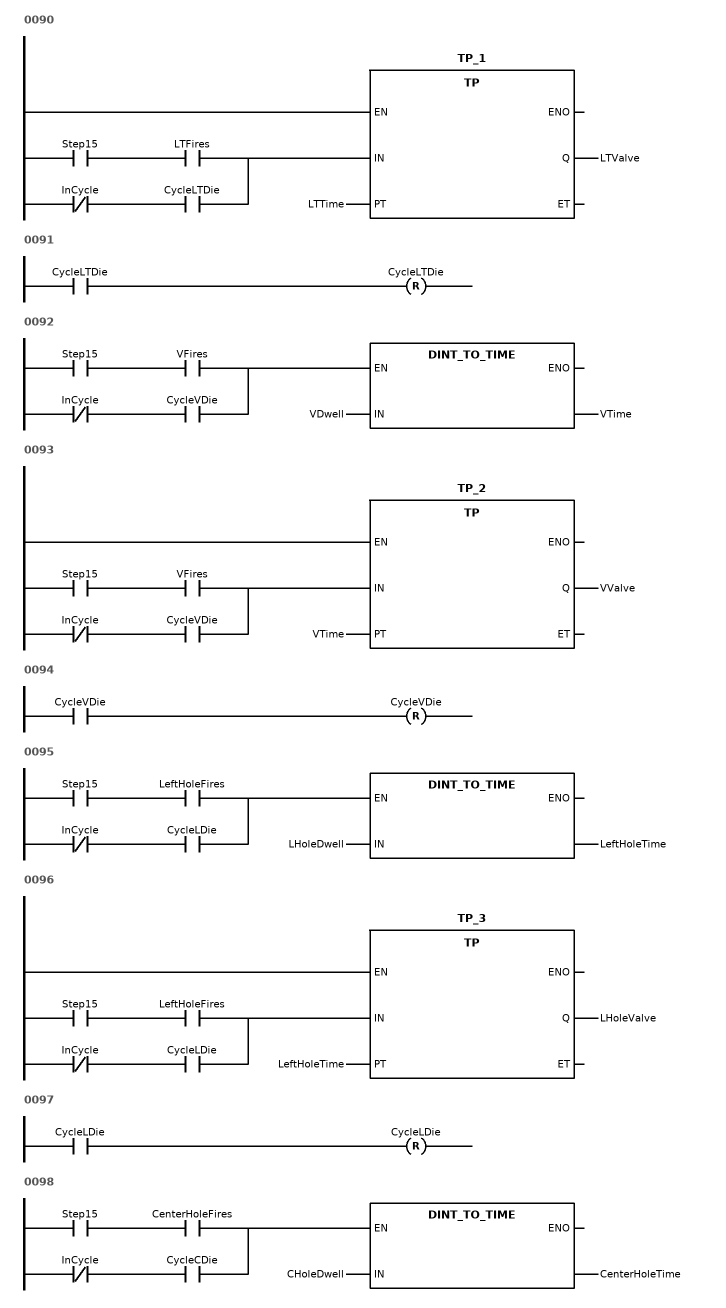
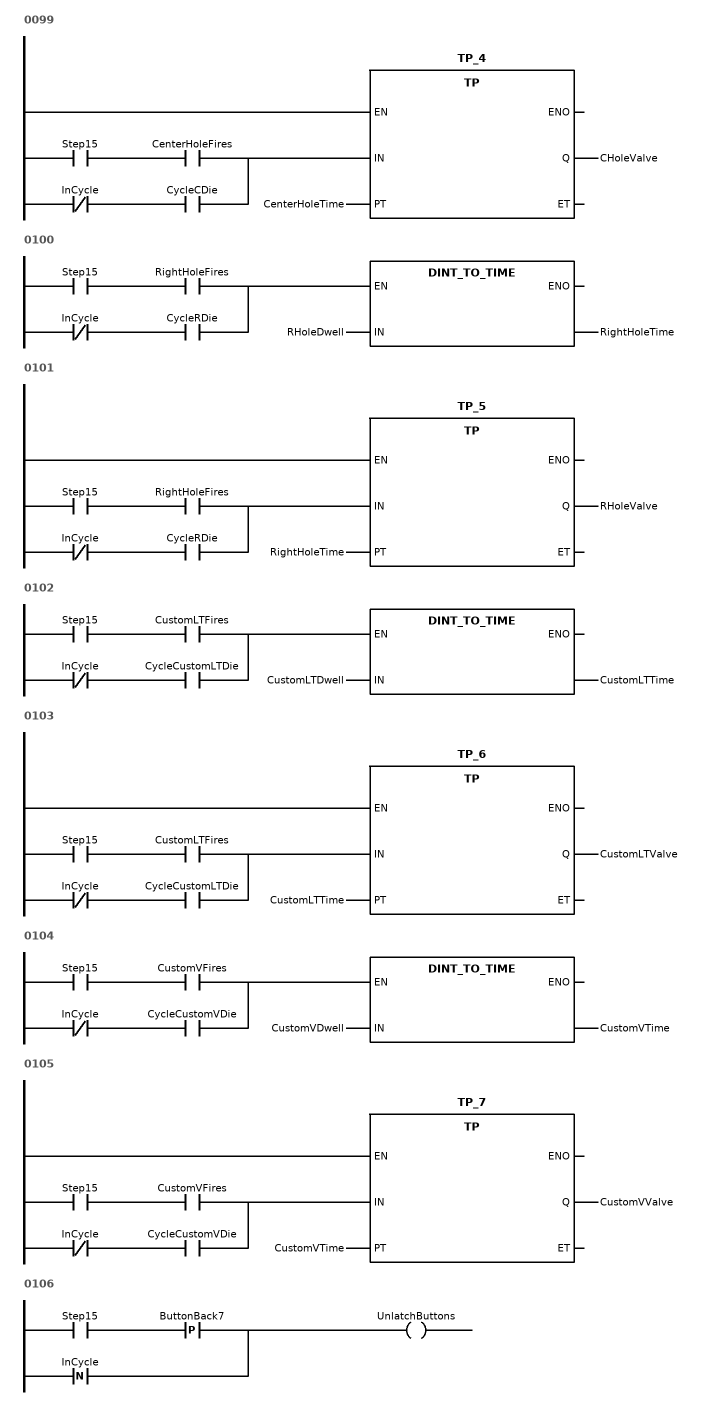
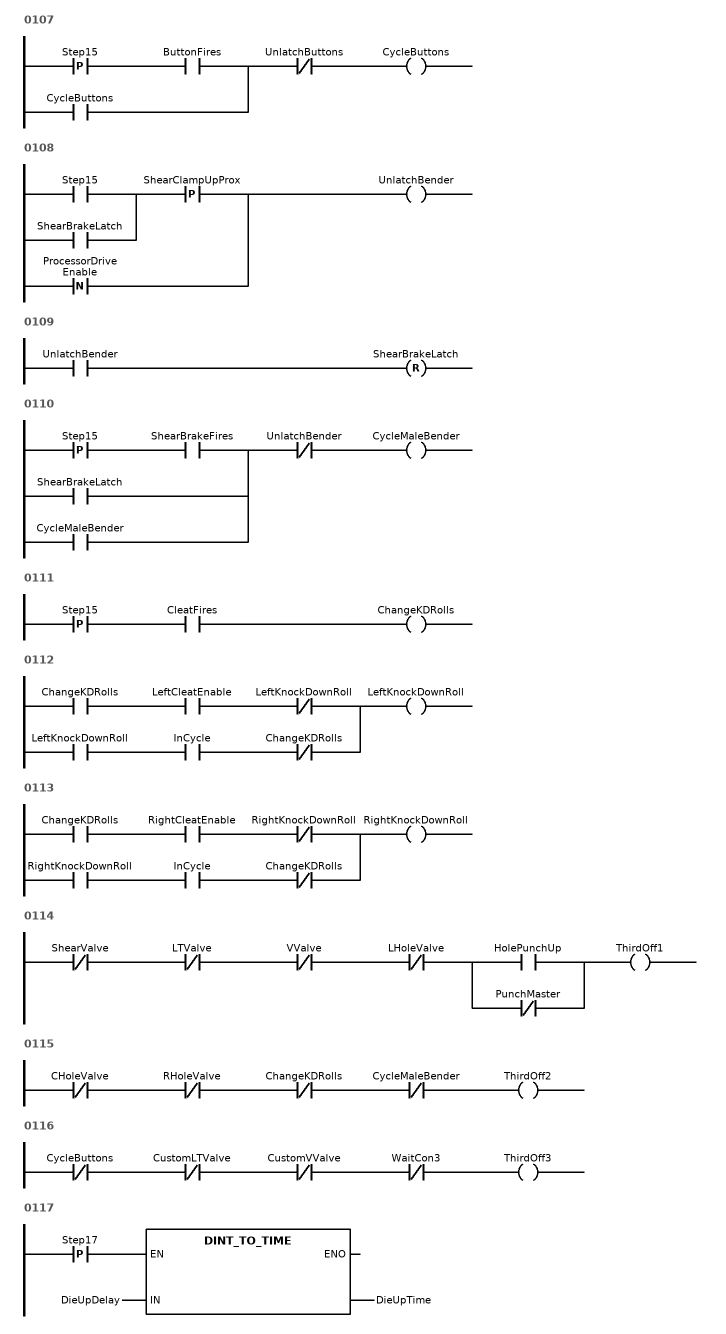
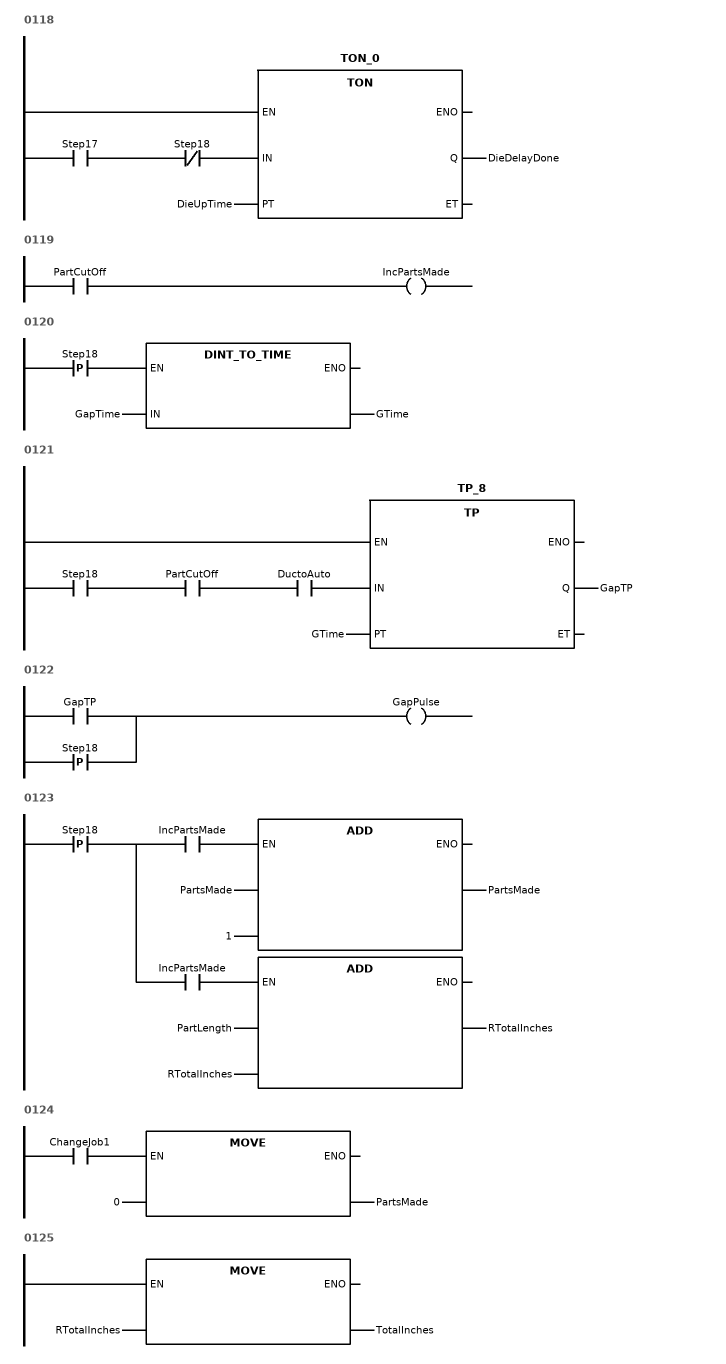
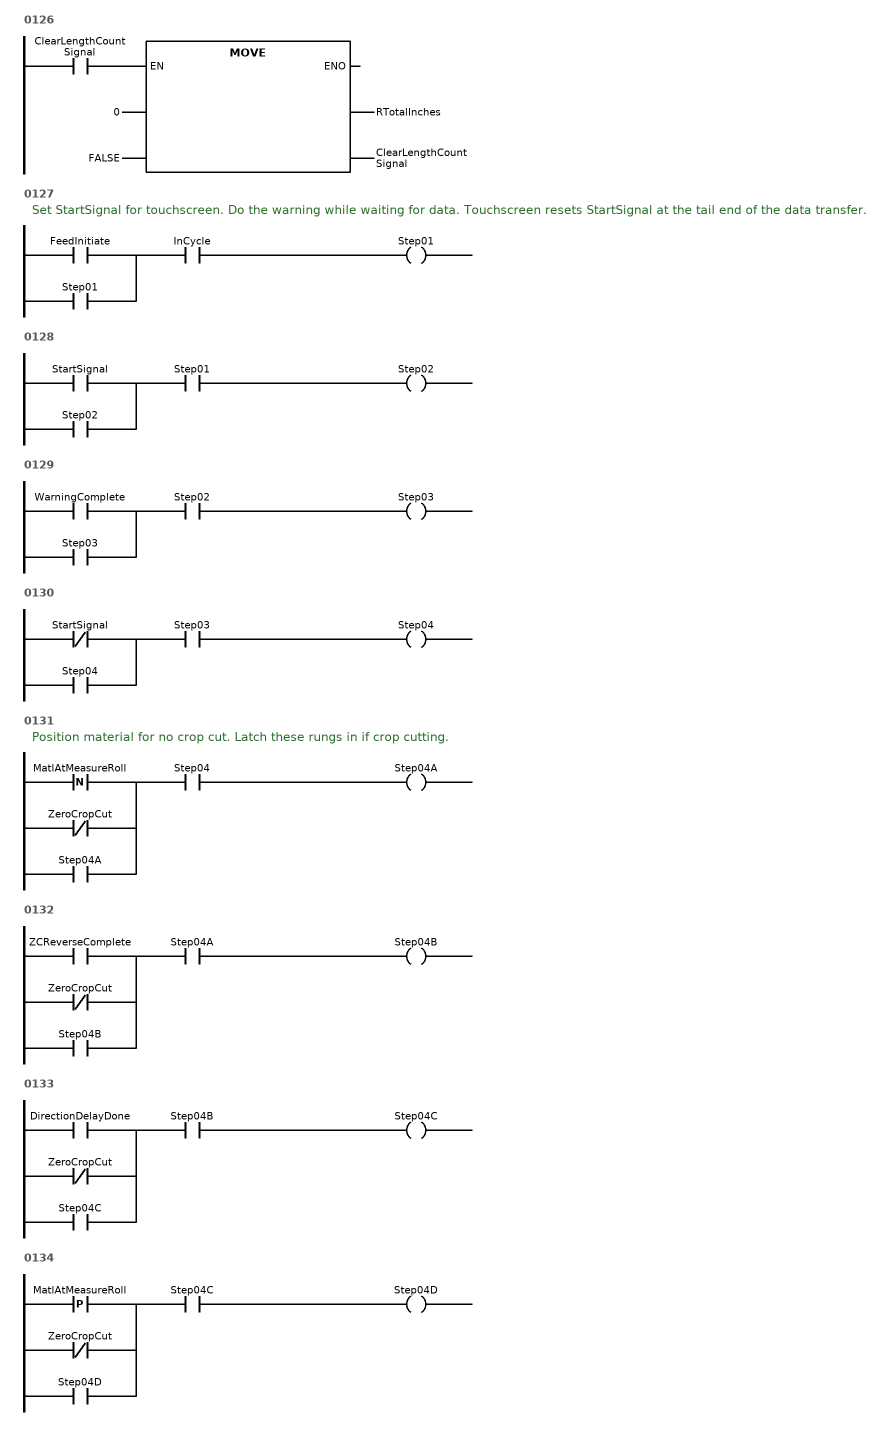
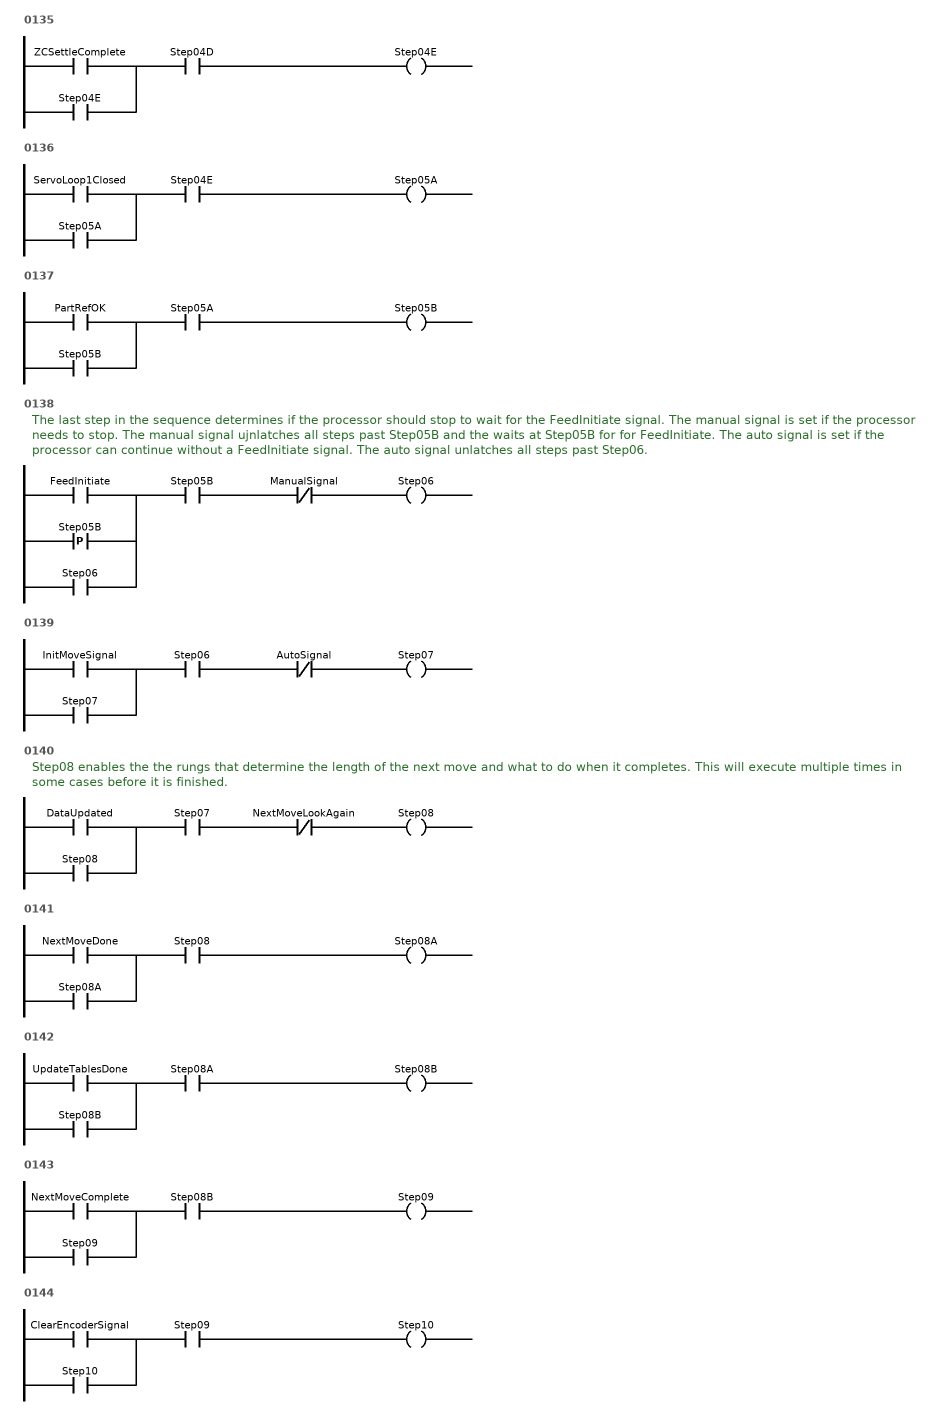
